% RSLogix 500 project I2P Hands-On 4 - Mitch.RSS, saved by version 10.00.00.00 %
PROJECT "UNTITLED"    % processor: Bul.1763 MicroLogix 1100 Series B %

PROGRAM FILES
  LAD 2   15 rungs

DATA FILES
  O0 OUTPUT  4 elements
  I1 INPUT  6 elements
  S2 STATUS  66 elements
  B3 BINARY  1 elements
  T4 TIMER  1 elements
  C5 COUNTER  1 elements
  R6 CONTROL  1 elements
  N7 INTEGER  1 elements
  F8 FLOAT  1 elements

LADDER 2
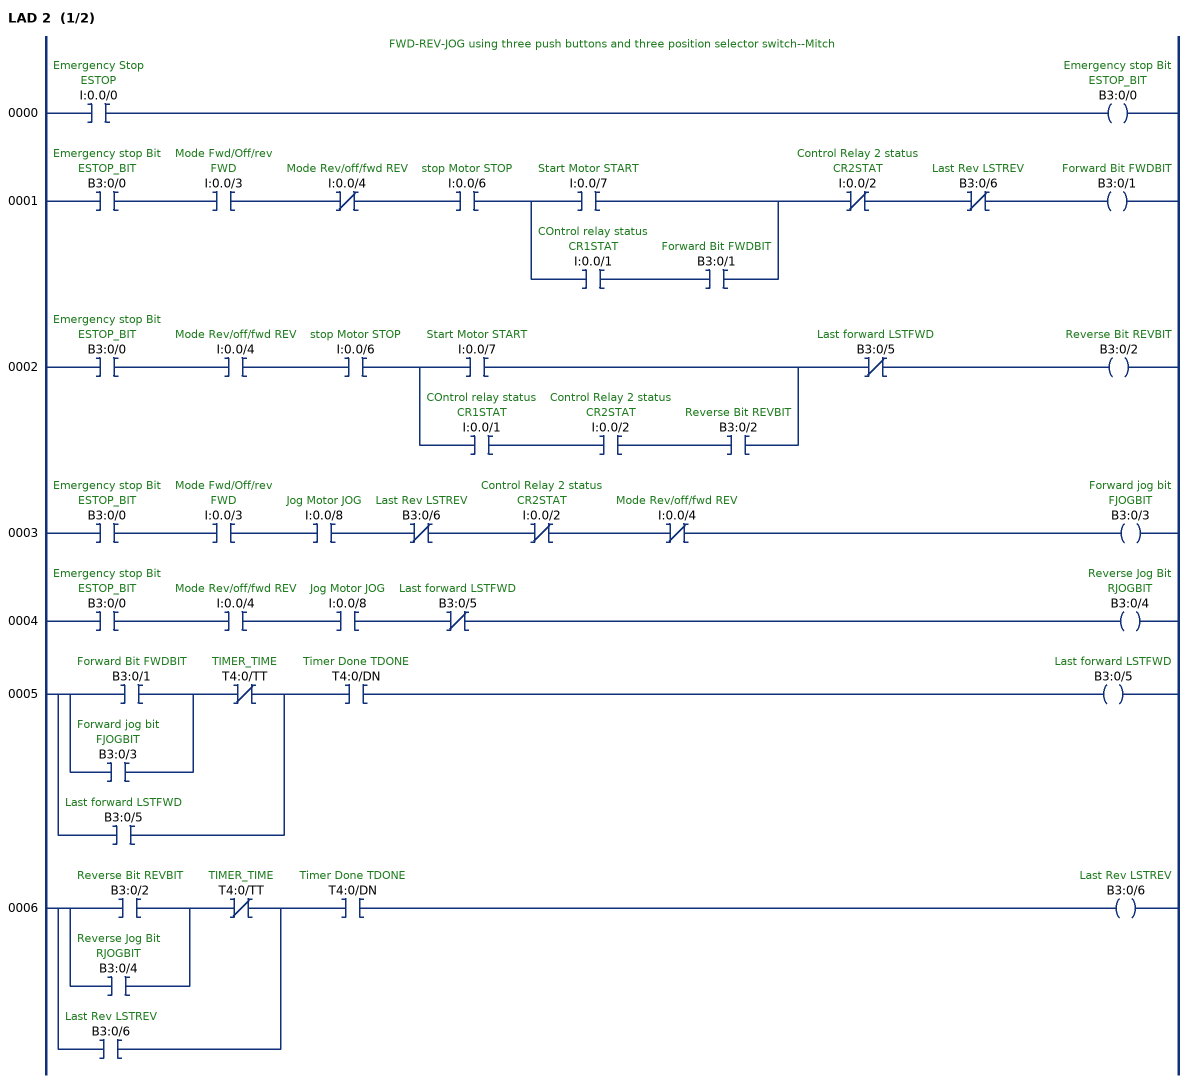
% Rung: 0 %
% FWD-REV-JOG using three push buttons and three position selector switch--Mitch %
SOR XIC I:0.0/0 OTE B3:0/0 EOR
%   I:0.0/0  ESTOP  "Emergency Stop" %
%   B3:0/0  ESTOP_BIT  "Emergency stop Bit" %
% Rung: 1 %
SOR XIC B3:0/0 XIC I:0.0/3 XIO I:0.0/4 XIC I:0.0/6 BST XIC I:0.0/7 NXB XIC I:0.0/1 XIC B3:0/1 BND XIO I:0.0/2 XIO B3:0/6 OTE B3:0/1 EOR
%   B3:0/0  ESTOP_BIT  "Emergency stop Bit" %
%   I:0.0/3  FWD  "Mode Fwd/Off/rev" %
%   I:0.0/4  REV  "Mode Rev/off/fwd" %
%   I:0.0/6  STOP  "stop Motor" %
%   I:0.0/7  START  "Start Motor" %
%   I:0.0/1  CR1STAT  "COntrol relay status" %
%   B3:0/1  FWDBIT  "Forward Bit" %
%   I:0.0/2  CR2STAT  "Control Relay 2 status" %
%   B3:0/6  LSTREV  "Last Rev" %
% Rung: 2 %
SOR XIC B3:0/0 XIC I:0.0/4 XIC I:0.0/6 BST XIC I:0.0/7 NXB XIC I:0.0/1 XIC I:0.0/2 XIC B3:0/2 BND XIO B3:0/5 OTE B3:0/2 EOR
%   B3:0/0  ESTOP_BIT  "Emergency stop Bit" %
%   I:0.0/4  REV  "Mode Rev/off/fwd" %
%   I:0.0/6  STOP  "stop Motor" %
%   I:0.0/7  START  "Start Motor" %
%   I:0.0/1  CR1STAT  "COntrol relay status" %
%   I:0.0/2  CR2STAT  "Control Relay 2 status" %
%   B3:0/2  REVBIT  "Reverse Bit" %
%   B3:0/5  LSTFWD  "Last forward" %
% Rung: 3 %
SOR XIC B3:0/0 XIC I:0.0/3 XIC I:0.0/8 XIO B3:0/6 XIO I:0.0/2 XIO I:0.0/4 OTE B3:0/3 EOR
%   B3:0/0  ESTOP_BIT  "Emergency stop Bit" %
%   I:0.0/3  FWD  "Mode Fwd/Off/rev" %
%   I:0.0/8  JOG  "Jog Motor" %
%   B3:0/6  LSTREV  "Last Rev" %
%   I:0.0/2  CR2STAT  "Control Relay 2 status" %
%   I:0.0/4  REV  "Mode Rev/off/fwd" %
%   B3:0/3  FJOGBIT  "Forward jog bit" %
% Rung: 4 %
SOR XIC B3:0/0 XIC I:0.0/4 XIC I:0.0/8 XIO B3:0/5 OTE B3:0/4 EOR
%   B3:0/0  ESTOP_BIT  "Emergency stop Bit" %
%   I:0.0/4  REV  "Mode Rev/off/fwd" %
%   I:0.0/8  JOG  "Jog Motor" %
%   B3:0/5  LSTFWD  "Last forward" %
%   B3:0/4  RJOGBIT  "Reverse Jog Bit" %
% Rung: 5 %
SOR BST BST XIC B3:0/1 NXB XIC B3:0/3 BND XIO T4:0/TT NXB XIC B3:0/5 BND XIC T4:0/DN OTE B3:0/5 EOR
%   B3:0/1  FWDBIT  "Forward Bit" %
%   B3:0/3  FJOGBIT  "Forward jog bit" %
%   T4:0/TT  TIMER_TIME %
%   B3:0/5  LSTFWD  "Last forward" %
%   T4:0/DN  TDONE  "Timer Done" %
% Rung: 6 %
SOR BST BST XIC B3:0/2 NXB XIC B3:0/4 BND XIO T4:0/TT NXB XIC B3:0/6 BND XIC T4:0/DN OTE B3:0/6 EOR
%   B3:0/2  REVBIT  "Reverse Bit" %
%   B3:0/4  RJOGBIT  "Reverse Jog Bit" %
%   T4:0/TT  TIMER_TIME %
%   B3:0/6  LSTREV  "Last Rev" %
%   T4:0/DN  TDONE  "Timer Done" %

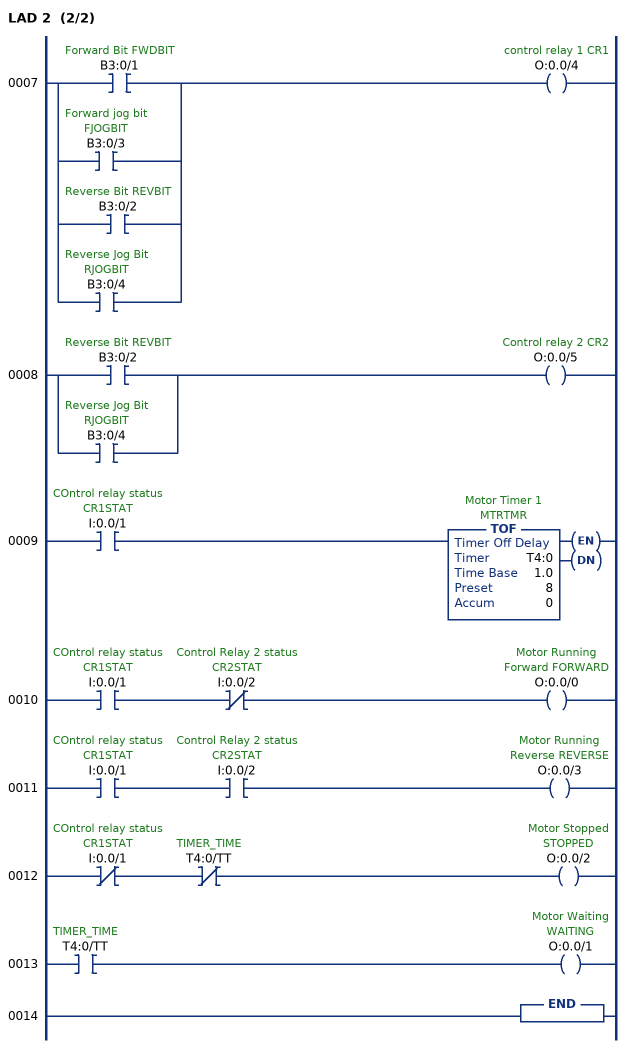
% Rung: 7 %
SOR BST BST XIC B3:0/1 NXB XIC B3:0/3 BND NXB BST XIC B3:0/2 NXB XIC B3:0/4 BND BND OTE O:0.0/4 EOR
%   B3:0/1  FWDBIT  "Forward Bit" %
%   B3:0/3  FJOGBIT  "Forward jog bit" %
%   B3:0/2  REVBIT  "Reverse Bit" %
%   B3:0/4  RJOGBIT  "Reverse Jog Bit" %
%   O:0.0/4  CR1  "control relay 1" %
% Rung: 8 %
SOR BST XIC B3:0/2 NXB XIC B3:0/4 BND OTE O:0.0/5 EOR
%   B3:0/2  REVBIT  "Reverse Bit" %
%   B3:0/4  RJOGBIT  "Reverse Jog Bit" %
%   O:0.0/5  CR2  "Control relay 2" %
% Rung: 9 %
SOR XIC I:0.0/1 TOF T4:0 1.0 8 0 EOR
%   I:0.0/1  CR1STAT  "COntrol relay status" %
%   T4:0  MTRTMR  "Motor Timer 1" %
% Rung: 10 %
SOR XIC I:0.0/1 XIO I:0.0/2 OTE O:0.0/0 EOR
%   I:0.0/1  CR1STAT  "COntrol relay status" %
%   I:0.0/2  CR2STAT  "Control Relay 2 status" %
%   O:0.0/0  FORWARD  "Motor Running Forward" %
% Rung: 11 %
SOR XIC I:0.0/1 XIC I:0.0/2 OTE O:0.0/3 EOR
%   I:0.0/1  CR1STAT  "COntrol relay status" %
%   I:0.0/2  CR2STAT  "Control Relay 2 status" %
%   O:0.0/3  REVERSE  "Motor Running Reverse" %
% Rung: 12 %
SOR XIO I:0.0/1 XIO T4:0/TT OTE O:0.0/2 EOR
%   I:0.0/1  CR1STAT  "COntrol relay status" %
%   T4:0/TT  TIMER_TIME %
%   O:0.0/2  STOPPED  "Motor Stopped" %
% Rung: 13 %
SOR XIC T4:0/TT OTE O:0.0/1 EOR
%   T4:0/TT  TIMER_TIME %
%   O:0.0/1  WAITING  "Motor Waiting" %
% Rung: 14 %
SOR END EOR

DATA TABLE (non-zero values as saved)
DATA T4
% .PRE .ACC %
% T4:0 % 8 0
